FUNCTION F_5Args : INT VAR_INPUT a : INT; b : INT; c : INT; d : INT; e : INT; END_VAR

F_5Args := a + b + c + d + e;

END_FUNCTION

(* stored: Version 1.1.0.1, ProductVersion 3.1.4024.16
   POU F_5Args: Id {8a0c5ce6-0d2a-4701-8807-d359c246cb9b}, SpecialFunc None *)
